FUNCTION_BLOCK LockingRelay EXTENDS Object
VAR_INPUT
END_VAR
VAR_OUTPUT
END_VAR
VAR
  _clk: BOOL;
  r_clk: R_TRIG;
END_VAR

PROPERTY clk : BOOL
SET
r_clk(CLK:=clk);
IF r_clk.Q THEN
  _clk := TRUE;
ELSIF NOT clk THEN
  _clk := FALSE;
END_IF
END_SET
END_PROPERTY

PROPERTY q : BOOL
GET
q := _clk;
END_GET
END_PROPERTY

PROPERTY reset : BOOL
SET
IF reset THEN
  _clk := FALSE;
END_IF
END_SET
END_PROPERTY

END_FUNCTION_BLOCK

(* stored: Version 1.1.0.1, ProductVersion 3.1.4022.18
   POU LockingRelay: Id {12380fa4-bd87-480a-ae60-f4eb89316508}, SpecialFunc None
   Property clk: Id {ee0c0626-704a-4f08-bf99-09c57a59d5fa}
   Set Set: Id {2d5ae0a2-c8df-41a8-ac5f-f5614d1e5fe9}
   Property q: Id {2c523e14-85e7-4951-9898-90dfbbe8beda}
   Get Get: Id {60e82940-38ed-4c54-8bea-f925007193ff}
   Property reset: Id {fb134051-2622-4fb0-84e8-0daf166880b1}
   Set Set: Id {df089b9f-542a-4a11-b9fc-af2f7e455db2} *)
